(* Logix 5000 project; controller ECE119L_AnalogTest 5069-L306ERM rev 32.11; software revision 32.04 *)

TASK MainTask (continuous, watchdog 500 ms) : MainProgram

MODULES
   Local : 5069-L306ERM (5069 0, rev 32.11)
      Analog_inputs : vendor 1 type 115 code 314 (5069 4, rev 2.1, StandardDataDriven RPI 100 ms)
      Analog_Output : vendor 1 type 115 code 320 (5069 5, rev 2.1, StandardDataDriven RPI 80 ms)
      Digital_Output : 5069-OB16 (5069 2, rev 3.1, StandardDataDriven RPI 5 ms)
      Analog_In : vendor 1 type 115 code 314 (5069 3, rev 2.1, StandardDataDriven RPI 100 ms)
      Digital_Inputs : vendor 1 type 7 code 391 (5069 1, rev 2.1, StandardDataDriven RPI 5 ms)
END_MODULES

VAR_GLOBAL   (* controller tags *)
   LCD_Screen : ALIAS FOR Local:5:O.Ch00.Data;
   Potentiometer : ALIAS FOR Local:4:I.CJCh00.Temperature;
   Red_Led : ALIAS FOR Local:2:O.Pt08.Data;
END_VAR

PROGRAM MainProgram   (* main routine MainRoutine *)

ROUTINE MainRoutine   (* ladder *)
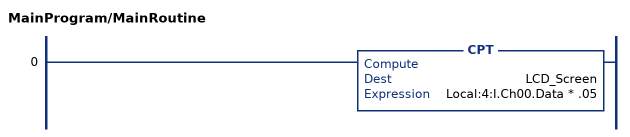
   0: CPT(LCD_Screen,Local:4:I.Ch00.Data * .05);
END_ROUTINE
END_PROGRAM
